// TIA Portal V20 export
// export: Created 2026-04-11T06:02:30.4816256Z, ExportSetting WithDefaults, DisplayName Totally Integrated Automation Portal, DisplayVersion V20, DisplayName TIA Portal Openness, DisplayVersion V20, DisplayName TIA Portal Version Control Interface, DisplayVersion V20, DisplayName STEP 7 Professional, DisplayVersion V20, DisplayName STEP 7 Safety, DisplayVersion V20, DisplayName WinCC Basic/Comfort/Advanced, DisplayVersion V20, DisplayName WinCC Unified, DisplayVersion V20
TYPE "udtHMI_FlowTotalizer"
// stored: IsFailsafeCompliant false
   STRUCT
      bPB_ResetResult : Bool;
      bPBEN_ResetResult : Bool;
      bPB_Pause : Bool;
      bPBEN_Pause : Bool;
      rOutScaledValue : Real;
      HMI_AnalogInput { S7_SetPoint := 'True'} : "udtHMI_AnalogInput";
   END_STRUCT;
END_TYPE
